(* Schneider Machine Expert - Basic project SimulationHMIPLC, file version 1.8.0.0 *)
(* ProjectInformations: Name=Yeni proje *)

HARDWARE
  Cpu 0: TM221ME16T/G
  EthernetConfiguration: NetworkName=M221, IpAllocationMode=FixedAddress, IpAddress=0.0.0.0, SubnetMask=0.0.0.0
  SerialLineConfiguration: Baud=Baud19200, Parity=ParityEven, DataBits=DataBits8, StopBits=StopBits1, PhysicalMedium=PhysicalMediumRs485, TransmissionMode=TransmissionModeModbusRtu, SlaveId=1, Addressing=SlaveAddressing
  MastTask: UsePeriodScanMode=false, PeriodScan=100
  FastTask: Period=255
  CpuBehavior: StartingMode=StartAsPreviousState, AutoSaveRamOnEeprom=true, WatchdogPeriod=250

SYMBOLS  (address, symbol, comment, settings)

POU Yeni POU
  (* SectionNumber=1 *)

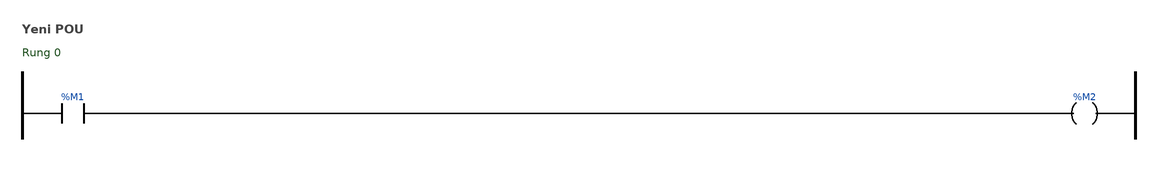

// Rung 0
  LD %M1
  ST %M2
  // as ST:
  //   %M2 := %M1;
